PROGRAM MAIN
VAR
	ipot1OutputJeanPaul AT %Q* :INT;
END_VAR

 ArrayStorage();
 Case_Chase();
 StructureTesting();
 
 ipot1OutputJeanPaul := gvl.iPot1;

END_PROGRAM

(* stored: Version 1.1.0.1, ProductVersion 3.1.4024.12
   POU MAIN: Id {752f5c4e-fd2e-4946-8870-50266f7ca74a}, SpecialFunc None *)
